// TIA Portal V19 export
TYPE "C701_VAR_IF_VNU_TYPIC"
   STRUCT
      STO { ExternalAccessible := 'False'; ExternalVisible := 'False'; ExternalWritable := 'False'} : Bool;   // Storing algemeen ventilatie unit
   END_STRUCT;
END_TYPE
